FUNCTION_BLOCK FB_FT_PIWL2 (* Basic Function Block Type *)
  (* Standard: 61499-2 *)
  (* Version 0.0, 2011-07-20, 4DIAC-IDE, 4DIAC-Consortium *)
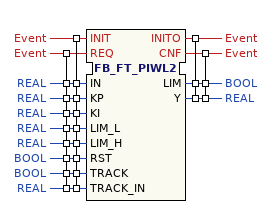
  EVENT_INPUT
    INIT WITH IN, KP, KI, LIM_L, LIM_H, RST, TRACK, TRACK_IN; (* Initialization Request *)
    REQ WITH IN, KP, LIM_L, KI, LIM_H, RST, TRACK, TRACK_IN; (* Normal Execution Request *)
  END_EVENT
  EVENT_OUTPUT
    INITO WITH LIM, Y; (* Initialization Confirm *)
    CNF WITH LIM, Y; (* Execution Confirmation *)
  END_EVENT
  VAR_INPUT
    IN : REAL; (* Input *)
    KP : REAL := 1.0; (* Amplification factor for proportional controller *)
    KI : REAL := 1.0; (* Amplification factor for integrator *)
    LIM_L : REAL := -1.0E38; (* lowest possible output range *)
    LIM_H : REAL := 1.0E38; (* highest possible output range *)
    RST : BOOL; (* Resets integrator to 0 *)
    TRACK : BOOL; (* Switch tracking on or off *)
    TRACK_IN : REAL; (* Tracking input *)
  END_VAR
  VAR_OUTPUT
    LIM : BOOL; (* Returns true if output limit is active *)
    Y : REAL; (* Output *)
  END_VAR
  VAR
    tx : DWORD; (* system time *)
    tc : REAL; (* difference between last and actual system time *)
    t_last : DWORD; (* last system time *)
    in_last : REAL; (* last input *)
    i : REAL; (* variable to calculate Y *)
    p : REAL; (* variable to calculate Y *)
  END_VAR
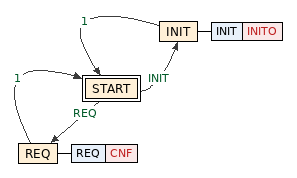
  EC_STATES
    START; (* Initial State *)
    INIT : INIT -> INITO; (* Initialization *)
    REQ : REQ -> CNF; (* Normal execution *)
  END_STATES
  EC_TRANSITIONS
    START TO INIT := INIT;
    INIT TO START := 1;
    START TO REQ := REQ;
    REQ TO START := 1;
  END_TRANSITIONS
  ALGORITHM INIT IN ST: (* Initialization algorithm *)
in_last := IN;
t_last := T_PLC_US();
i := 0.0;
tc := 0.0;
  END_ALGORITHM
  ALGORITHM REQ IN ST: (* Normally executed algorithm *)
IF RST THEN
	in_last := IN;
	t_last := T_PLC_US();
	i := 0.0;
	tc := 0.0;
ELSE
	(* read last cycle time in Microseconds *)
	tx := T_PLC_US();
	tc := DWORD_TO_REAL(tx - t_last);
	t_last := tx;

	(* calculate proportional part *)
	p := KP * IN;

	(* run integrator *)

	IF TRACK THEN
		i := TRACK_IN - p;
	ELSE
		i := (IN + in_last) * 5.0E-7 * KI * tc + i;
		in_last := IN;
	END_IF
	(* calculate output Y *)
	Y := p + i;

	(* check output for limits *)
	IF Y >= LIM_H THEN
		Y := LIM_H;
		IF KI <> 0.0 THEN
			i := LIM_H - p;
		ELSE
			i := 0.0;
		END_IF;
		LIM := TRUE;
	ELSIF Y <= LIM_L THEN
		Y := LIM_L;
		IF KI <> 0.0 THEN
			i := LIM_L - p;
		ELSE
			i := 0.0;
		END_IF;
		LIM := TRUE;
	ELSE
		LIM := FALSE;
	END_IF;
END_IF;
  END_ALGORITHM
END_FUNCTION_BLOCK
